(* IEC 61131-3 sources: JaccoSigma/tempclass/Class/MyPW, 1 file *)

(* ---- MyPW.st ---- *)
(*!
<Class
	Name               = "MyPW"
	Revision           = "0.0"
	RealtimeTask       = "false"
	CyclicTask         = "false"
	BackgroundTask     = "false"
	Sigmatek           = "false"
	OSInterface        = "false"
	HighPriority       = "false"
	Automatic          = "false"
	UpdateMode         = "Prescan"
	SharedCommandTable = "true"
	Objectsize         = "(284,120)">
	<Channels>
		<Server Name="ClassSvr" Visualized="true" Initialize="false" WriteProtected="false" Retentive="false"/>
	</Channels>
</Class>
*)
MyPW : CLASS
  //Servers:
	ClassSvr 	: SvrChCmd_DINT;
  //Clients:
  //Variables:
  //Functions:
  //Tables:
	FUNCTION @STD
		VAR_OUTPUT
			ret_code	: CONFSTATES;
		END_VAR;
	FUNCTION GLOBAL TAB @CT_;
END_CLASS;
